PROGRAM MAIN
VAR
END_VAR

END_PROGRAM

(* stored: Version 1.1.0.1
   POU MAIN: Id {4f701a96-5522-4ba4-ac52-498eee76cf05} *)
